{attribute 'GeneratedUsingTerminal: KL9999'}
{attribute addProperty BoxType "KL9999"}
{attribute addProperty Id "Channel_1AT %Q*Channel_126527430"}
{attribute addProperty CRC "2047911926"}
{attribute addProperty Size "0"}
TYPE KL9999_7A10A7F6 :
STRUCT
	{attribute addProperty Name "Channel_1"}
	Channel_1 : Channel_12652743;
END_STRUCT
END_TYPE

(* stored: Version 1.2.0.0, ProductVersion 3.1.4024.9
   DUT KL9999_7A10A7F6: Id {82e8adf3-c7f9-4f70-b1d6-fbf4e23fc7ed} *)
